TYPE ST_SYSTEM_SafetyStatus :
STRUCT
	bSafetyRelayOK					: BOOL;
	bEStopButtonPressed				: BOOL;
	bEmergencyCircuitOK				: BOOL;
	bGuardDoorOK						: BOOL;
	bMotorDriversOK					: BOOL;
	bSafetyOK						: BOOL;			(* All systems Go! *)

END_STRUCT
END_TYPE

(* stored: Version 1.1.0.1
   DUT ST_SYSTEM_SafetyStatus: Id {558cfa0f-6d4d-42cd-b2a3-22e44fe6f43a} *)
